GLOBALCONSTANTS AID_AO (* Animation object attribute ids *)
  (* Standard: 61499-1; Description: Copyright (c) 2023 HR Agrartechnik GmbH This program and the accompanying materials are made available under the terms of the Eclipse Public License 2.0 which is available at https://www.eclipse.org/legal/epl-2.0/ SPDX-License-Identifier: EPL-2.0 *)
  (* Version 1.0, 2026-06-20, Franz Höpfinger, HR Agrartechnik GmbH *)
  PACKAGE isobus::UT::Q::const::AID;
  VAR_GLOBAL CONSTANT
    WIDTH : USINT := USINT#1; (* 1: AID_AO_WIDTH - Width in pixels. *)
    HEIGHT : USINT := USINT#2; (* 2: AID_AO_HEIGHT - Height in pixels. *)
    REFRESHINT : USINT := USINT#3; (* 3: AID_AO_REFRESHINT *)
    VALUE : USINT := USINT#4; (* 4: AID_AO_VALUE - Current value. *)
    ENABLED : USINT := USINT#5; (* 5: AID_AO_ENABLED - 0 = Stopped, 1 = Animating. *)
    FICHILDINDEX : USINT := USINT#6; (* 6: AID_AO_FICHILDINDEX *)
    LACHILDINDEX : USINT := USINT#7; (* 7: AID_AO_LACHILDINDEX *)
    DEFCHILDINDEX : USINT := USINT#8; (* 8: AID_AO_DEFCHILDINDEX *)
    OBJECTS : USINT := USINT#9; (* 9: AID_AO_OBJECTS - OPTIONS - Bit 0: Animation Sequence (0=Single Shot, 1=Loop). Bits 1-2: Disabled Behaviour (0=Pause, 1=Reset to First, 2=Default Object, 3=Blank). *)
  END_VAR
END_GLOBALCONSTANTS
